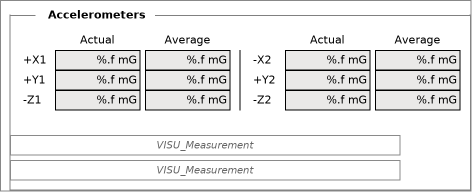
VISUALIZATION VISU_TelemetryAccelerometers  // 472x192
VAR_IN_OUT
	ref : TelemetryAccelerometers;
    widget : TelemetryAccelerometersWidget;
END_VAR
    Polyline (155,15) (470,15) (470,190) (10,190) (10,15) (35,15)
    Label (45,5 115x20), "Accelerometers"
    Label (20,50 35x20), "+X1"
    Rectangle (55,50 85x20), "%.f mG", text variable: ref.tube.X1plus.actual.milliG.value, colour toggle: ref.tube.X1plus.error
    Label (20,70 35x20), "+Y1"
    Rectangle (55,70 85x20), "%.f mG", text variable: ref.tube.Y1plus.actual.milliG.value, colour toggle: ref.tube.Y1plus.error
    Label (20,90 35x20), "-Z1"
    Rectangle (55,90 85x20), "%.f mG", text variable: ref.tube.Z1minus.actual.milliG.value, colour toggle: ref.tube.Z1minus.error
    Label (250,50 35x20), "-X2"
    Rectangle (285,50 85x20), "%.f mG", text variable: ref.tube.X2minus.actual.milliG.value, colour toggle: ref.tube.X2minus.error
    Label (250,70 35x20), "+Y2"
    Rectangle (285,70 85x20), "%.f mG", text variable: ref.tube.Y2plus.actual.milliG.value, colour toggle: ref.tube.Y2plus.error
    Label (250,90 35x20), "-Z2"
    Rectangle (285,90 85x20), "%.f mG", text variable: ref.tube.Z2minus.actual.milliG.value, colour toggle: ref.tube.Z2minus.error
    Frame (10,135 390x20)
        shows VISU_Measurement(widget := widget.tubeX)
    Line (240,110) (240,50)
    Frame (10,160 390x20)
        shows VISU_Measurement(widget := widget.tubeY)
    Rectangle (145,50 85x20), "%.f mG", text variable: ref.tube.X1plus.average.milliG.value, colour toggle: ref.tube.X1plus.error
    Rectangle (145,90 85x20), "%.f mG", text variable: ref.tube.Z1minus.average.milliG.value, colour toggle: ref.tube.Z1minus.error
    Rectangle (145,70 85x20), "%.f mG", text variable: ref.tube.Y1plus.average.milliG.value, colour toggle: ref.tube.Y1plus.error
    Label (55,30 85x20), "Actual"
    Label (145,30 85x20), "Average"
    Label (375,30 85x20), "Average"
    Label (285,30 85x20), "Actual"
    Rectangle (375,50 85x20), "%.f mG", text variable: ref.tube.X2minus.average.milliG.value, colour toggle: ref.tube.X2minus.error
    Rectangle (375,90 85x20), "%.f mG", text variable: ref.tube.Z2minus.average.milliG.value, colour toggle: ref.tube.Z2minus.error
    Rectangle (375,70 85x20), "%.f mG", text variable: ref.tube.Y2plus.average.milliG.value, colour toggle: ref.tube.Y2plus.error
END_VISUALIZATION

(* stored: Version 1.1.0.1, ProductVersion 3.1.4019.2
   Visu VISU_TelemetryAccelerometers: Id {b1efd739-8ccd-4481-9da7-31127be02ad2} *)
